(* CoDeSys 2.3.9.50 project: 2A.pr6 *)
(* Libraries: STANDARD.LB6 5.6.98 12:03:02 *)

(* POU MAIN, LD *)
PROGRAM MAIN
VAR
	Forward AT %QX0.0: BOOL;
	Reverse AT %QX0.1: BOOL;
	SwitchA AT %IX0.0: BOOL;
	SwitchB AT %IX0.1: BOOL;
END_VAR
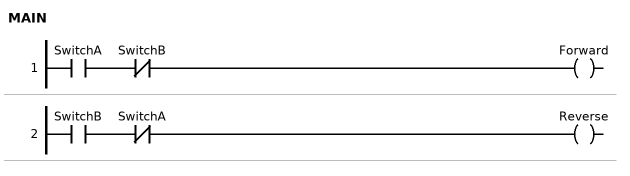
_LD_ (* Ladder Diagram *)
NETWORK 1
	[SwitchA] - [/SwitchB] --- (Forward)
NETWORK 2
	[SwitchB] - [/SwitchA] --- (Reverse)
_END_LD_
(* the same logic as Structured Text *)
(* Network 1 *)
Forward := SwitchA AND NOT SwitchB;
(* Network 2 *)
Reverse := SwitchB AND NOT SwitchA;
END_PROGRAM

(* Visualisation Q2A
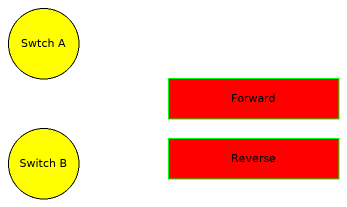
ellipse at (130,110)-(201,181): text "Swtch A"; alarm colour if %IX0.0; toggles %ix0.0
ellipse at (130,230)-(201,301): text "Switch B"; alarm colour if %IX0.1; toggles %IX0.1
rectangle at (290,180)-(461,221): text "Forward"; invisible if %QX0.0; toggles %QX0.0
rectangle at (290,240)-(461,281): text "Reverse"; invisible if %QX0.1; toggles %QX0.1
*)
